FUNCTION scaling : LREAL
VAR_INPUT
	fInput : LREAL;
	fScalingNum : LREAL;
	fScalingDenum : LREAL;
END_VAR

Scaling := fInput * (fScalingNum / fScalingDenum);

END_FUNCTION

(* stored: Version 1.1.0.1, ProductVersion 3.1.4024.12
   POU scaling: Id {9728d94c-cc60-407b-8e4d-6483ead09ef5}, SpecialFunc None *)
